// TwinCAT 3 PLC project Untitled1
// ProgramVersion: 3.1.4023.0
// libraries:
//   Tc2_Standard, * (Beckhoff Automation GmbH)
//   Tc2_System, * (Beckhoff Automation GmbH)
//   Tc2_Utilities, * (Beckhoff Automation GmbH)
//   Tc3_Module, * (Beckhoff Automation GmbH)
// project tree:
//   DUTs/ E_EventType.TcDUT, ST_Event.TcDUT, WeekDay.TcDUT
//   GVLs/ GVL.TcGVL
//   / PlcTask.TcTTO
//   POUs/ I_PersistentStorage.TcIO, Eventlogger.TcPOU, MAIN.TcPOU, POU.TcPOU, UpdateEventTimeStampWithSystemTime.TcPOU, FB_CSVPersistentEventStorage.TcPOU
// real-time tasks:
//   TASK PlcTask: cycle T#10ms, priority 20, ADS port 350
//   TASK PlcTask1: cycle T#10ms, priority 21, ADS port 351

CONFIGURATION Untitled1
    RESOURCE PLC ON TwinCAT3
        TASK PlcTask(INTERVAL := T#10ms, PRIORITY := 20);
        PROGRAM MAIN WITH PlcTask : MAIN;
    END_RESOURCE
END_CONFIGURATION

// ---- DUTs/E_EventType.TcDUT
{attribute 'qualified_only'}
{attribute 'strict'}
{attribute 'to string'}
TYPE E_EventType :
(
	Alarm,
	Message
);
END_TYPE

// ---- DUTs/ST_Event.TcDUT
TYPE ST_Event :
STRUCT
	eEventType: E_EventType;
	eEventSeverity: TcEventSeverity;
	nEventIdentity: UDINT;
	sEventText: STRING(255);
	dtTimeStamp: DT;
END_STRUCT
END_TYPE

// ---- DUTs/WeekDay.TcDUT
//{attribute 'qualified_only'}
//{attribute 'strict'}
TYPE WeekDay :
(
	Monday := 1,
	Tuesday := 2,
	Wednesday := 3,
	Thursday := 4,
	Friday := 5,
	Saturday := 6,
	Sunday := 0
);
END_TYPE

// ---- GVLs/GVL.TcGVL
{attribute 'qualified_only'}
VAR_GLOBAL
	vaerde: INT;
	
END_VAR

// ---- POUs/I_PersistentStorage.TcIO
INTERFACE I_PersistentStorage

METHOD StoreEvent
VAR_INPUT
	stEvent: ST_Event;
END_VAR
END_METHOD

END_INTERFACE

// ---- POUs/MAIN.TcPOU
PROGRAM MAIN
VAR
	//stThisIsOurFirstInstanceOfAStructure: ST_Event;
	bBoolean: BOOL:= FALSE;
	//n: INT;
	//trigger: BOOL;
	
	
	//LocalSystemTime: FB_LocalSystemTime();
		//timeStruct: TIMESTRUCT;
	CSVPersistentEventStorage: FB_CSVPersistentEventStorage;	
	Eventlogger:Eventlogger(CSVPersistentEventStorage);
	
	//SQLPersistentEventStorage: SQLPersistentEventStorage;
	//Eventlogger2:Eventlogger(SQLPersistentEventStorage);
	
	eEventType: E_EventType:=E_EventType.Alarm ;
	eEventSeverity: TcEventSeverity:=TcEventSeverity.Critical;
	nEventIdentity: UDINT:=1;
	sEventText: STRING(255):= 'Allvarligt fel';

	testLogger: Eventlogger;
	fbNy: POU;
	
END_VAR

IF NOT bBoolean THEN
	Eventlogger.AddEvent(eEventType:= eEventType,eEventSeverity:= eEventSeverity,nEventIdentity:=nEventIdentity,sEventText:=sEventText);
	
	bBoolean:= TRUE;
END_IF


CSVPersistentEventStorage();

//LocalSystemTime(bEnable:=TRUE,systemTime=> timeStruct);

//stThisIsOurFirstInstanceOfAStructure.dtTimeStamp := SYSTEMTIME_TO_DT(TIMESTR:=timeStruct);
//stThisIsOurFirstInstanceOfAStructure.sEventText:= 'TEST';

END_PROGRAM

// ---- POUs/FB_CSVPersistentEventStorage.TcPOU
FUNCTION_BLOCK FB_CSVPersistentEventStorage IMPLEMENTS I_PersistentStorage

VAR
	
	fileOpen: FB_FileOpen:=(sPathName:='c:\Events.log',nMode:= FOPEN_MODEAPPEND OR FOPEN_MODETEXT );
	fileClose: FB_FileClose;
	filePuts: FB_FilePuts;
	eWriteState: (FILE_OPEN_TRIGGER,FILE_OPEN, WAIT_FOR_EVENT, WRITE_EVENT_TRIGGER,WRITE_EVENT, FILE_CLOSE_TRIGGER, FILE_CLOSE, ERROR);
	stEventWrittenToFile: ST_Event;
	
	CsvString:T_MaxString;
	
END_VAR

CASE eWriteState OF
	FILE_OPEN_TRIGGER:
				fileOpen(bExecute:=TRUE);
				eWriteState:= FILE_OPEN;
	FILE_OPEN:
				fileOpen(bExecute:=FALSE);
				IF fileOpen.bError THEN
					eWriteState:= ERROR;
				ELSIF NOT fileOpen.bBusy AND fileOpen.hFile <> 0 THEN
					eWriteState := WAIT_FOR_EVENT;		
				END_IF
	WAIT_FOR_EVENT:
		//Do Nothing
	WRITE_EVENT_TRIGGER:
		CsvString := CreateCsvString(stEvent:=stEventWrittenToFile);
		
		filePuts(bExecute:= TRUE, sLine:=CsvString,hFile:=fileOpen.hFile );
		eWriteState := WRITE_EVENT;
				
	WRITE_EVENT:
			filePuts(bExecute:=FALSE);
			IF filePuts.bError THEN
					eWriteState:= ERROR;
				ELSIF NOT filePuts.bBusy  THEN
					eWriteState := FILE_CLOSE_TRIGGER;		
				END_IF
	FILE_CLOSE_TRIGGER:
		fileClose(bExecute:=TRUE,hFile:=fileOpen.hFile);
				eWriteState := FILE_CLOSE;
	FILE_CLOSE:
		fileClose(bExecute:=FALSE);
		IF fileClose.bError THEN
			eWriteState:= ERROR;
		ELSIF NOT fileClose.bBusy THEN
			eWriteState:=	FILE_OPEN_TRIGGER;
		END_IF
	ERROR:
	//Error Code here
	
END_CASE

METHOD CreateCsvString : T_MaxString
VAR_INPUT
	stEvent: REFERENCE TO ST_Event;
	
END_VAR
VAR
	Tempstring: T_MaxString;
END_VAR
Tempstring:= TO_STRING(stEvent.eEventType);
Tempstring:=CONCAT(STR1:= Tempstring, STR2:= ',');
Tempstring:=CONCAT(STR1:= Tempstring, STR2:= TO_STRING(stEvent.eEventSeverity));
Tempstring:=CONCAT(STR1:= Tempstring, STR2:= ',');
Tempstring:=CONCAT(STR1:= Tempstring, STR2:= TO_STRING(stEvent.nEventIdentity));
Tempstring:=CONCAT(STR1:= Tempstring, STR2:= ',');
Tempstring:=CONCAT(STR1:= Tempstring, STR2:= TO_STRING(stEvent.sEventText));
Tempstring:=CONCAT(STR1:= Tempstring, STR2:= ',');
Tempstring:=CONCAT(STR1:= Tempstring, STR2:= TO_STRING(stEvent.dtTimeStamp));
Tempstring:=CONCAT(STR1:= Tempstring, STR2:= '$n');

CreateCsvString:= Tempstring;
END_METHOD

{warning 'add method implementation '}
METHOD StoreEvent
VAR_INPUT
	stEvent	: ST_Event;
END_VAR
//Implement code here
IF eWriteState =  WAIT_FOR_EVENT THEN
	eWriteState:= WRITE_EVENT_TRIGGER;
	stEventWrittenToFile:=stEvent;

END_IF
END_METHOD

END_FUNCTION_BLOCK

// ---- POUs/Eventlogger.TcPOU
FUNCTION_BLOCK Eventlogger
VAR
	Eventbuffer: ARRAY [1..MAXIMUM_NUMBER_OF_EVENTS] OF ST_Event;
	CurrentEventNumber : INT :=0;
	_PersistentEventStorage: I_PersistentStorage;
	
END_VAR
VAR CONSTANT
	MAXIMUM_NUMBER_OF_EVENTS: INT:=100;
END_VAR

METHOD PUBLIC AddEvent : BOOL
VAR_INPUT
	eEventType: E_EventType;
	eEventSeverity: TcEventSeverity;
	nEventIdentity: UDINT;
	sEventText: STRING(255);
END_VAR
IF NOT IsEventBufferFull() THEN
		CurrentEventNumber := CurrentEventNumber +1;
		Eventbuffer[CurrentEventNumber].eEventType:= eEventType;
		Eventbuffer[CurrentEventNumber].eEventSeverity:=eEventSeverity;
		Eventbuffer[CurrentEventNumber].nEventIdentity:=nEventIdentity;
		Eventbuffer[CurrentEventNumber].sEventText:=sEventText;
	UpdateEventTimeStampWithSystemTime(stEvent:= Eventbuffer[CurrentEventNumber]);	

AddEvent:=TRUE;
	ELSE
		AddEvent:=FALSE;	
	END_IF
	
	
	//Here we want to store the event persistently
	_PersistentEventStorage.StoreEvent(stEvent:=Eventbuffer[CurrentEventNumber]);
END_METHOD

METHOD FB_init : BOOL
VAR_INPUT
	bInitRetains : BOOL; // if TRUE, the retain variables are initialized (warm start / cold start)
	bInCopyCode : BOOL;  // if TRUE, the instance afterwards gets moved into the copy code (online change)
	iPersistentStorage: I_PersistentStorage;
	
END_VAR
_PersistentEventStorage:=iPersistentStorage;
END_METHOD

METHOD PRIVATE IsEventBufferFull : BOOL
VAR_INPUT
END_VAR
IsEventBufferFull:= (CurrentEventNumber+1 > MAXIMUM_NUMBER_OF_EVENTS);
END_METHOD

END_FUNCTION_BLOCK

// ---- POUs/UpdateEventTimeStampWithSystemTime.TcPOU
FUNCTION UpdateEventTimeStampWithSystemTime
VAR_INPUT
	stEvent: REFERENCE TO ST_Event;
 
END_VAR
VAR
	//timeStruct: TIMESTRUCT;
	 //LocalSystemTime: FB_LocalSystemTime();
	 fbGetsytstemtime: GETSYSTEMTIME;
	 filetime: T_FILETIME;
END_VAR


//LocalSystemTime(bEnable:=TRUE,systemTime=> timeStruct);
//timeStruct;
fbGetsytstemtime(timeLoDW=> filetime.dwLowDateTime, timeHiDW=> filetime.dwHighDateTime);//SYSTEMTIME_TO_DT(TIMESTR:=timeStruct);
stEvent.dtTimeStamp:= FILETIME_TO_DT(filetime);

END_FUNCTION

// ---- POUs/POU.TcPOU
FUNCTION_BLOCK POU
VAR_INPUT
END_VAR
VAR_OUTPUT
END_VAR
VAR
END_VAR

END_FUNCTION_BLOCK
